// Hand-written example of what the protoc code generator would produce
// for a "Motor1" device DDATA message (DATA mode — alias-only, no names).
//
// Aliases match the DBIRTH schema (FB_Motor1_Birth):
//   alias 1 — Speed       (UInt32, rpm)
//   alias 2 — Running     (Boolean)
//   alias 3 — Temperature (Float, °C)
//
// DATA messages omit metric names (sName := '') to save bandwidth. The host
// resolves alias → name from the preceding DBIRTH.
//
// Usage:
//   IF tPublish.Q AND fbSession.bOnline THEN
//     fbMotor1Data.Build(F_GetUnixTimestampMs(), fbSession.GetNextSeq(), nSpeed, bRunning, fTemp);
//     fbSession.Publish(sDataTopic, fbMotor1Data.Buffer, fbMotor1Data.Length);
//   END_IF
FUNCTION_BLOCK FB_Motor1_Data
VAR
	_aBuf		: ARRAY[0..127] OF BYTE;	// smaller — no metric names in DATA mode
	_fbPayload	: FB_SparkplugPayload;
END_VAR

// FB body intentionally empty — all logic is in Build().

PROPERTY Buffer : POINTER TO BYTE
GET
Buffer := _fbPayload.Buffer;
END_GET
END_PROPERTY

// Encodes the DDATA payload (alias-only, no metric names).
// nSeq must come from FB_SparkplugSession.GetNextSeq() immediately before publishing.
METHOD Build : BOOL
VAR_INPUT
	nTimestamp		: ULINT;
	nSeq			: ULINT;
	nSpeed			: UDINT;
	bRunning		: BOOL;
	fTemperature	: REAL;
END_VAR
_fbPayload.Init(ADR(_aBuf), SIZEOF(_aBuf));
_fbPayload.WriteHeader(nTimestamp, nSeq);
// DATA mode: sName := '' — alias is written, name is omitted
_fbPayload.WriteUInt32Metric('', 1, E_SparkplugDataType.UInt32,  nSpeed);
_fbPayload.WriteBoolMetric  ('', 2, E_SparkplugDataType.Boolean, bRunning);
_fbPayload.WriteFloatMetric ('', 3, E_SparkplugDataType.Float,   fTemperature);
Build := NOT _fbPayload.HasError;
END_METHOD

PROPERTY Length : UDINT
GET
Length := _fbPayload.Length;
END_GET
END_PROPERTY

END_FUNCTION_BLOCK

(* stored: Version 1.1.0.1
   POU FB_Motor1_Data: Id {cc000002-0000-0000-0000-000000000000}, SpecialFunc None
   Property Buffer: Id {cc000002-0000-0000-0000-000000000002}
   Get Get: Id {cc000002-0000-0000-0000-000000000003}
   Method Build: Id {cc000002-0000-0000-0000-000000000001}
   Property Length: Id {cc000002-0000-0000-0000-000000000004}
   Get Get: Id {cc000002-0000-0000-0000-000000000005} *)
